GLOBALCONSTANTS IG4_Source_Addresses (* Industry Group 4 specific source addresses *)
  (* Standard: 61499-1 *)
  (* Version 1.0, 2026-06-29, Franz Höpfinger, Demmler Andreas Fahrzeugbau *)
  PACKAGE isobus::pgn::const;
  VAR_GLOBAL CONSTANT
    SA_RESERVED_128 : BYTE := 128; (* Source Address: thru 207 are reserved for future assignment by SAE - Used for dynamic address *)
    SA_RESERVED_208 : BYTE := 208; (* Source Address: thru 227 are reserved for future assignment - Used for individual preassigned *)
    SA_PROPULSION_SENSOR_HUB_GATEWAY_1 : BYTE := 228; (* Source Address: Propulsion Sensor Hub & Gateway #1 - The first device that interfaces with *)
    SA_PROPULSION_SENSOR_HUB_GATEWAY_2 : BYTE := 229; (* Source Address: Propulsion Sensor Hub & Gateway #2 - The second device that interfaces with *)
    SA_PROPULSION_SENSOR_HUB_GATEWAY_3 : BYTE := 230; (* Source Address: Propulsion Sensor Hub & Gateway #3 - The third device that interfaces with *)
    SA_PROPULSION_SENSOR_HUB_GATEWAY_4 : BYTE := 231; (* Source Address: Propulsion Sensor Hub & Gateway #4 - The fourth device that interfaces with *)
    SA_TRANSMISSION_3 : BYTE := 232; (* Source Address: Transmission #3 - The Transmission ECU for the third transmission within a system *)
    SA_TRANSMISSION_4 : BYTE := 233; (* Source Address: Transmission #4 - The Transmission ECU for the fourth transmission within a *)
    SA_TRANSMISSION_5 : BYTE := 234; (* Source Address: Transmission #5 - The Transmission ECU for the fifth transmission within a system *)
    SA_TRANSMISSION_6 : BYTE := 235; (* Source Address: Transmission #6 - The Transmission ECU for the sixth transmission within a system *)
    SA_DISPLAY_1_FOR_PROTECTION_SYSTEM_FOR_MARINE_ENGINES : BYTE := 236; (* Source Address: Display #1 for Protection System for Marine Engines - The first ecu that provides *)
    SA_PROTECTION_SYSTEM_FOR_MARINE_ENGINES : BYTE := 237; (* Source Address: Protection System for Marine Engines - The first ecu that controls the Protection *)
    SA_ALARM_SYSTEM_CONTROL_1_FOR_MARINE_ENGINES : BYTE := 238; (* Source Address: Alarm System Control #1 for Marine Engines - The first ecu that controls the *)
    SA_ENGINE_3 : BYTE := 239; (* Source Address: Engine #3 - The Engine ECU for the third engine within a system. *)
    SA_ENGINE_4 : BYTE := 240; (* Source Address: Engine #4 - The Engine ECU for the fourth engine within a system. *)
    SA_ENGINE_5 : BYTE := 241; (* Source Address: Engine #5 - The Engine ECU for the fifth engine within a system. *)
    SA_MARINE_DISPLAY_1 : BYTE := 242; (* Source Address: Marine Display #1 - The first Marine Display for an engine. *)
    SA_MARINE_DISPLAY_2 : BYTE := 243; (* Source Address: Marine Display #2 - The second Marine Display for an engine. *)
    SA_MARINE_DISPLAY_3 : BYTE := 244; (* Source Address: Marine Display #3 - The third Marine Display for an engine. *)
    SA_MARINE_DISPLAY_4 : BYTE := 245; (* Source Address: Marine Display #4 - The fourth Marine Display for an engine. *)
    SA_MARINE_DISPLAY_5 : BYTE := 246; (* Source Address: Marine Display #5 - The fifth Marine Display for an engine. *)
    SA_MARINE_DISPLAY_6 : BYTE := 247; (* Source Address: Marine Display #6 - The sixth Marine Display for an engine. *)
  END_VAR
END_GLOBALCONSTANTS
